FUNCTION_BLOCK EventLogger
VAR_INPUT
END_VAR
VAR_OUTPUT
END_VAR
VAR
END_VAR

END_FUNCTION_BLOCK

(* stored: Version 1.1.0.1, ProductVersion 3.1.4024.12
   POU EventLogger: Id {59da52f9-b004-4470-a33e-2933fcde4a2b}, SpecialFunc None *)
